// TIA Portal V17 export
// export: Created 2024-03-30T11:15:07.1727506Z, ExportSetting WithDefaults, DisplayName Totally Integrated Automation Portal, DisplayVersion V17, DisplayName TIA Portal Openness, DisplayVersion V17, DisplayName TIA Portal Version Control Interface, DisplayVersion V17, DisplayName STEP 7 Professional, DisplayVersion V17, DisplayName STEP 7 Safety, DisplayVersion V17, DisplayName WinCC Advanced, DisplayVersion V17
TYPE "typ_Axis"
// stored: IsFailsafeCompliant false
   STRUCT
      x_Start_Positioning : Bool;
      x_Reference : Bool;
      x_Referenced : Bool;
      x_Position_Reached : Bool;
      di_Target_Position : DInt;
      di_Increment : DInt;
      di_Actual_Position : DInt := 0;
      i_PWM : Int;
      Config : "typ_Axis_Data";
   END_STRUCT;
END_TYPE
